PROGRAM FastPRG_1
VAR

END_VAR

(*__________________________________________________________________________________________________
¦	
¦	Vistaprint Schweiz GmbH
¦	CH - 8401 Winterthur
¦
¦	www.vistaprint.ch - info@vistaprint.ch
¦___________________________________________________________________________________________________

Function desription:
call of all controller (FUB) for the fast task class.


History:
Version		Date			Author		Comment
---------------------------------------------------------------------------------------------------
0.00.1		25.05.2013		AVME/KVO	Start history


___________________________________________________________________________________________________*)


// -----------------------------------------------------------------------------------------------
// Initialize the PLC Parameter and check the PLC health
// -----------------------------------------------------------------------------------------------
IF (g_uinStartProzess=0) THEN
	g_uinStartProzess:=1; // For StartUp order

END_IF
// -----------------------------------------------------------------------------------------------


// -----------------------------------------------------------------------------------------------
// The host system is downloading all parameter at startup. 
// bolPlcStartupDone will be set to true after the Host is done with the initialization
// -----------------------------------------------------------------------------------------------
IF (g_uinStartProzess=c_uinCntTaskClass) THEN
	g_uinStartProzess := 11; // For StartUp order
END_IF
// -----------------------------------------------------------------------------------------------


// -----------------------------------------------------------------------------------------------
// Start PLC code initialization
// -----------------------------------------------------------------------------------------------
IF (g_uinStartProzess=(10+c_uinCntTaskClass)) THEN
	
	// init	
	g_uinStartProzess := 21; // For StartUp order
END_IF
// -----------------------------------------------------------------------------------------------


// -----------------------------------------------------------------------------------------------
// Normal Run mode after1 all the initialization is done
// -----------------------------------------------------------------------------------------------
IF (g_uinStartProzess>=(20+c_uinCntTaskClass)) THEN
	;
END_IF
// -----------------------------------------------------------------------------------------------

END_PROGRAM

(* stored: Version 1.1.0.1, ProductVersion 3.1.0.25
   POU FastPRG_1: Id {cef9ae2e-c547-4599-8a76-ee84fec7c7c9} *)
